{attribute 'no_explicit_call' := 'Do not call this FB directly!'}
FUNCTION_BLOCK FB_Command IMPLEMENTS ICommand
VAR
	_Result		   : ST_Result;
	_SequenceState : DINT;
END_VAR

PROPERTY Busy : BOOL
GET
Busy := _Result.Busy;
END_GET
SET
_Result.Busy := Busy;
END_SET
END_PROPERTY

PROPERTY Done : BOOL
GET
Done := _Result.Done;
END_GET
SET
_Result.Done := Done;
END_SET
END_PROPERTY

PROPERTY Error : BOOL
GET
Error := _Result.Error;
END_GET
SET
_Result.Error := Error;
END_SET
END_PROPERTY

PROPERTY ErrorId : DINT
GET
ErrorId := _Result.ErrorId;
END_GET
SET
_Result.ErrorId := ErrorId;
END_SET
END_PROPERTY

PROPERTY Sequence : DINT
GET
Sequence := _SequenceState;
END_GET
SET
_SequenceState := Sequence;
END_SET
END_PROPERTY

METHOD Start : ICommand
VAR_INPUT
END_VAR
_SequenceState	:= 0;
_Result.Done	:= FALSE;
_Result.Busy	:= TRUE;
_Result.Error	:= FALSE;
_Result.ErrorId := 0;
Start			:= This^;
END_METHOD

END_FUNCTION_BLOCK

(* stored: Version 1.1.0.1, ProductVersion 3.1.4024.12
   POU FB_Command: Id {249951de-6bd4-4b91-9e01-c50dc6584630}, SpecialFunc None
   Folder ICommand: Id {18b292a5-ab55-40fb-9c83-cf12fe1af791}
   Folder IResult: Id {88dfa4a4-87d0-44c9-b9c4-2683530fc236}
   Property Busy: Id {eb2116ce-7b80-498b-8fa3-24b72b6b1ab8}
   Get Get: Id {243d34d5-f54a-4d2b-a429-d629b4ff95c7}
   Set Set: Id {0b8649e0-f75b-4ff0-9c0c-a676c5419db2}
   Property Done: Id {145a12f9-563a-4476-9c36-5161e646eb3a}
   Get Get: Id {6fb4f4c4-5366-49dc-a465-da33934aafb2}
   Set Set: Id {489fe03f-2d29-4b97-9a89-b401cc3e0d1c}
   Property Error: Id {b861ea8d-2427-4bb9-aa8b-798798dee58c}
   Get Get: Id {f849cec0-1def-44c7-9730-338fdb0c7099}
   Set Set: Id {1746f02d-844c-48a1-a900-95b47611f1ec}
   Property ErrorId: Id {f732ec30-9827-422a-8e82-63bdacafdc65}
   Get Get: Id {c0d87b78-9e4f-491b-98c2-2192bb564786}
   Set Set: Id {64c4a577-3aed-470f-aa78-0d430bea7ac6}
   Property Sequence: Id {1895c768-df50-4383-9ff7-e5d178fa0e04}
   Get Get: Id {24049301-0a87-4e44-8100-e8010248d8c0}
   Set Set: Id {dc1400bc-3de2-460c-b3c8-e506839cbdca}
   Method Start: Id {24f98774-f64d-425b-bec3-a1db94820221} *)
